// TIA Portal project "SCDW_PlcProject" (V17)

(* hardware
DEVICE "PLC_1"  S7-1500 station
   slot 0: "导轨_0"  Rack  6ES7 590-1***0-0AA0
   slot 1: "PLC_1"  CPU 1513-1 PN  6ES7 513-1AL00-0AB0  V1.8
      slot 3: "CPU 显示_1"  6ES7591-1AA00-0AA0
      slot 32768: "PROFINET 接口_1"  X1
         slot 32769: "端口_1"  X1 P1
         slot 32770: "端口_2"  X1 P2
*)

// ===== PLC "PLC_1"  CPU 1513-1 PN =====

ORGANIZATION_BLOCK "Main"   // OB1, LAD, ProgramCycle
TITLE = "Main Program Sweep (Cycle)"
{ S7_Optimized_Access := 'TRUE' }
VERSION : 0.1
   VAR_INPUT
      Initial_Call : Bool;   // Initial call of this OB
      Remanence : Bool;   // =True, if remanent data are available
   END_VAR
BEGIN
END_ORGANIZATION_BLOCK